TYPE ST_OPCUA_Node_BOOL :
STRUCT
	NodeID				: ST_UANodeID;
	NodeHdl				: DWORD;
	SizeOfDataType		: UDINT;
	NodeAddInfo			: ST_UANodeAdditionalInfo;
	TargetVar			: POINTER TO BOOL;
END_STRUCT
END_TYPE

(* stored: Version 1.1.0.1, ProductVersion 3.1.4024.9
   DUT ST_OPCUA_Node_BOOL: Id {2a5c6952-97b8-4b47-ab61-fd030f38a35a} *)
